TYPE ST_Communication :
STRUCT
	Var1 : INT;
	Var2 : DINT;
	RecipeData: ST_RecipeData;
END_STRUCT
END_TYPE

(* stored: Version 1.1.0.1, ProductVersion 3.1.4018.2
   DUT ST_Communication: Id {b98b5717-5da6-45ac-b15e-f306aea34ed2} *)
